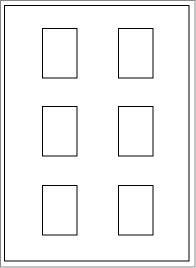
VISUALIZATION Carrinho_3  // 196x268
    RoundedRectangle (4,5 185x256)
    RoundedRectangle (35,36 50x35), angle 90, colour variable: GVL_P.corPosReator3[4].color
        OnMouseUp: execute { gvl.actReat:= 4; posCarrinho3(); }
        OnMouseUp: OpenDialog Dialog=ConfigPosicao_Reator_3, Parameters={bReator: , iOFnumber: , iSrlNumber: }, OpenModal=True, OpenCentered=True
    RoundedRectangle (111,36 50x35), angle 90, colour variable: GVL_P.corPosReator3[1].color
        OnMouseUp: OpenDialog Dialog=ConfigPosicao_Reator_3, Parameters={bReator: , iOFnumber: , iSrlNumber: }, OpenModal=True, OpenCentered=True
        OnMouseUp: execute { gvl.actReat:= 1; posCarrinho3(); }
    RoundedRectangle (111,114 50x35), angle 90, colour variable: GVL_P.corPosReator3[2].color
        OnMouseUp: execute { gvl.actReat:= 2; posCarrinho3(); }
        OnMouseUp: OpenDialog Dialog=ConfigPosicao_Reator_3, Parameters={bReator: , iOFnumber: , iSrlNumber: }, OpenModal=True, OpenCentered=True
    RoundedRectangle (35,114 50x35), angle 90, colour variable: GVL_P.corPosReator3[5].color
        OnMouseUp: execute { gvl.actReat:= 5; posCarrinho3(); }
        OnMouseUp: OpenDialog Dialog=ConfigPosicao_Reator_3, Parameters={bReator: , iOFnumber: , iSrlNumber: }, OpenModal=True, OpenCentered=True
    RoundedRectangle (111,193 50x35), angle 90, colour variable: GVL_P.corPosReator3[3].color
        OnMouseUp: execute { gvl.actReat:= 3; posCarrinho3(); }
        OnMouseUp: OpenDialog Dialog=ConfigPosicao_Reator_3, Parameters={bReator: , iOFnumber: , iSrlNumber: }, OpenModal=True, OpenCentered=True
    RoundedRectangle (35,193 50x35), angle 90, colour variable: GVL_P.corPosReator3[6].color
        OnMouseUp: execute { gvl.actReat:= 6; posCarrinho3(); }
        OnMouseUp: OpenDialog Dialog=ConfigPosicao_Reator_3, Parameters={bReator: , iOFnumber: , iSrlNumber: }, OpenModal=True, OpenCentered=True
END_VISUALIZATION

(* stored: Version 1.1.0.1, ProductVersion 3.1.4024.12
   Visu Carrinho_3: Id {2e742abe-b66f-4f07-b195-028f902585e1} *)
